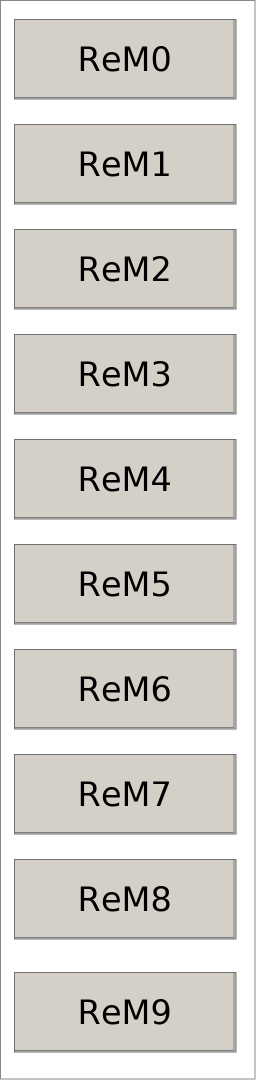
VISUALIZATION ReMList  // 256x1080
    Button (14,19 222x80), "ReM0", colour toggle: G_HMI.iReM =0
        p573394764: 16#FF00FF00
        OnMouseDown: execute { G_HMI.iReM  := 0; G_HMI.iMainFrame	:= 0; }
    Button (14,124 222x80), "ReM1", colour toggle: G_HMI.iReM =1
        p573394764: 16#FF00FF00
        OnMouseDown: execute { G_HMI.iReM  := 1; G_HMI.iMainFrame	:= 0; }
    Button (14,229 222x80), "ReM2", colour toggle: G_HMI.iReM =2
        p573394764: 16#FF00FF00
        OnMouseDown: execute { G_HMI.iReM  := 2; G_HMI.iMainFrame	:= 0; }
    Button (14,334 222x80), "ReM3", colour toggle: G_HMI.iReM =3
        p573394764: 16#FF00FF00
        OnMouseDown: execute { G_HMI.iReM  := 3; G_HMI.iMainFrame	:= 0; }
    Button (14,439 222x80), "ReM4", colour toggle: G_HMI.iReM =4
        p573394764: 16#FF00FF00
        OnMouseDown: execute { G_HMI.iReM  := 4; G_HMI.iMainFrame	:= 0; }
    Button (14,544 222x80), "ReM5", colour toggle: G_HMI.iReM =5
        p573394764: 16#FF00FF00
        OnMouseDown: execute { G_HMI.iReM  := 5; G_HMI.iMainFrame	:= 0; }
    Button (14,649 222x80), "ReM6", colour toggle: G_HMI.iReM =6
        p573394764: 16#FF00FF00
        OnMouseDown: execute { G_HMI.iReM  := 6; G_HMI.iMainFrame	:= 0; }
    Button (14,754 222x80), "ReM7", colour toggle: G_HMI.iReM =7
        p573394764: 16#FF00FF00
        OnMouseDown: execute { G_HMI.iReM  := 7; G_HMI.iMainFrame	:= 0; }
    Button (14,859 222x80), "ReM8", colour toggle: G_HMI.iReM =8
        p573394764: 16#FF00FF00
        OnMouseDown: execute { G_HMI.iReM  := 8; G_HMI.iMainFrame	:= 0; }
    Button (14,972 222x80), "ReM9", colour toggle: G_HMI.iReM =9
        p573394764: 16#FF00FF00
        OnMouseDown: execute { G_HMI.iReM  := 9; G_HMI.iMainFrame	:= 0; }
END_VISUALIZATION

(* stored: Version 1.1.0.1, ProductVersion 3.1.4024.12
   Visu ReMList: Id {2c1cc129-5e67-4f8a-b890-3aee9edbaf72} *)
